// TIA Portal V20 export
FUNCTION "Block_5" : Void   // FC5, FBD
{ S7_Optimized_Access := 'TRUE' }
// stored: SetENOAutomatically false
BEGIN

REGION Network 1
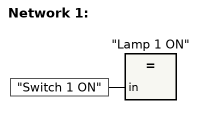
   "Lamp 1 ON" := "Switch 1 ON";
END_REGION
END_FUNCTION
